// TIA Portal V19 export
DATA_BLOCK "FlyingCarriage_PERS"   // DB136
{ DB_Accessible_From_OPC_UA := 'FALSE' }
// stored: DBAccessibleFromOPCUA false, MemoryReserve 100
   VAR RETAIN
      Parameter : "udt_FlyingCarriage_Parameter";
      FsParameter : "udt_FsParameter";
      SLS_Vel : LReal := 5000.0;
   END_VAR
BEGIN
   Parameter.PosTolerance := 0.1;
   Parameter.PosWindowDelay := T#200MS;
   Parameter.ZeroChk_SensorPosition := 57.32;
   Parameter.ZeroChk_PosTolerance := 3.0;
   Parameter.Limits.SwLimNegative := -5.0;
   Parameter.Limits.SwLimPositive := 1130.0;
   Parameter.Referencing.ApprochVelocity := 0.0;
   Parameter.Referencing.HomingVelocity := 0.0;
   Parameter.Referencing.HomePositionOffset := 0.0;
   Parameter.Referencing.HomePosition := 0.0;
   Parameter.Man.Vel := 5000.0;
   Parameter.Man.Acc := 3000.0;
   Parameter.Man.Dec := 5000.0;
   Parameter.Man.Jerk := 30000.0;
   Parameter.Aut.Vel := 50000.0;
   Parameter.Aut.Acc := 3000.0;
   Parameter.Aut.Dec := 3000.0;
   Parameter.Aut.Jerk := 20000.0;
   Parameter.Axis_Kv := 60.0;
   Parameter.Drive_Kp := 0.0;
   Parameter.Drive_Ki := 7.0;
   FsParameter.WorkMode := 4;
   FsParameter.Positions.HomePosition := 0.0;
   FsParameter.Positions.WorkEnablePosition := 0.0;
   FsParameter.Positions.ReturnEnablePosition := 0.0;
   FsParameter.Positions.StillCutPosition := 1080.0;
   FsParameter.ToolCycleTime := 0.0;
   FsParameter.FollowingErrorWindow := 0.1;
   FsParameter.DwellTimeErrorWindow := T#50MS;
   FsParameter.ErrorTimeout := T#10MS;
   FsParameter.BladeDetachValue := 0.0;
   FsParameter.BladeDetachVelocity := 5000.0;
   FsParameter.SyncDinamics.Acceleration := 3000.0;
   FsParameter.SyncDinamics.Jerk := 30000.0;
   FsParameter.SyncDinamics.ReturnVelocity := 50000.0;
   FsParameter.SyncDinamics.StartAdvanceSpace := 40.0;
   FsParameter.SyncDinamics.SyncLag := 2.0;
   FsParameter.SyncDinamics.ExtraSpeed := 1.0;
END_DATA_BLOCK
